VAR_GLOBAL
	InputArea	: ARRAY[0..15] OF BYTE;
	OutputArea	: ARRAY[0..15] OF BYTE;
END_VAR

(* stored: Version 1.1.0.1, ProductVersion 3.1.4024.6
   GVL GVL: Id {500f1e0c-03c6-40f0-9d2f-c532d7d3235a} *)
